// TIA Portal project "练习一视觉分拣" (V16)

(* hardware
DEVICE "S7-1200 station_1"  S7-1200 Station
   slot 0: "Rack_0"  S7-1200 Rack  Rack  V1.0
   slot 1: "PLC_1"  CPU 1214C DC/DC/Rly  6ES7 214-1HG40-0XB0  V4.4
DEVICE "HMI_1"  KTP700 Basic PN
   slot 0: "HMI_1"  KTP700 Basic PN  6AV2 123-2GB03-0AX0  16.0.0.0
   slot 1: "HMI_RT_1"  KTP700 Basic PN  6AV2 123-2GB03-0AX0  16.0.0.0
   slot 5: "HMI_1.IE_CP_1"  PROFINET Interface  16.0.0.0
      slot 1: "PROFINET Interface_1"  PROFINET Interface
         slot 1: "Port_1"  Port
*)

// ===== PLC "PLC_1"  CPU 1214C DC/DC/Rly =====

VAR_GLOBAL   // PLC tag table "默认变量表"
   "System_Byte" AT %MB1 : Byte;
   "FirstScan" AT %M1.0 : Bool;
   "DiagStatusUpdate" AT %M1.1 : Bool;
   "AlwaysTRUE" AT %M1.2 : Bool;
   "AlwaysFALSE" AT %M1.3 : Bool;
   "Clock_Byte" AT %MB0 : Byte;
   "Clock_10Hz" AT %M0.0 : Bool;
   "Clock_5Hz" AT %M0.1 : Bool;
   "Clock_2.5Hz" AT %M0.2 : Bool;
   "Clock_2Hz" AT %M0.3 : Bool;
   "Clock_1.25Hz" AT %M0.4 : Bool;
   "Clock_1Hz" AT %M0.5 : Bool;
   "Clock_0.625Hz" AT %M0.6 : Bool;
   "Clock_0.5Hz" AT %M0.7 : Bool;
END_VAR

VAR_GLOBAL   // PLC tag table "io"
   "启动信号" AT %I0.0 : Bool;
   "停止信号" AT %I0.1 : Bool;
   "复位信号" AT %I0.2 : Bool;
   "急停信号" AT %I0.3 : Bool;
   "左转到位i传感器" AT %I0.5 : Bool;
   "右转到位传感器" AT %I0.6 : Bool;
   "直行到位传感器" AT %I0.7 : Bool;
   "手动开关" AT %I1.0 : Bool;
   "自动开关" AT %I1.1 : Bool;
   "运行指示灯" AT %Q0.0 : Bool;
   "停止指示灯" AT %Q0.1 : Bool;
   "复位指示灯" AT %Q0.2 : Bool;
   "供料输送机" AT %Q0.3 : Bool;
   "直行电机" AT %Q0.4 : Bool;
   "左转电机" AT %Q0.5 : Bool;
   "右转电机" AT %Q0.6 : Bool;
   "产品原料分拣机" AT %Q0.7 : Bool;
   "产品基座分拣机" AT %Q1.0 : Bool;
   "产品盖分拣机" AT %Q1.1 : Bool;
   "物料生成器" AT %Q1.2 : Bool;
   "阻挡器" AT %Q1.3 : Bool;
   "视觉相机" AT %ID30 : DInt;
END_VAR

DATA_BLOCK "核心功能区"   // DB1
{ S7_Optimized_Access := 'TRUE' }
VERSION : 0.1
   VAR
      核心程序步 : Int;
      中间变量1 : Bool;
      中间变量2 : Bool;
      中间变量3 : Bool;
   END_VAR
BEGIN
END_DATA_BLOCK

DATA_BLOCK "FC程序视觉核心分拣区DB"   // DB2
{ S7_Optimized_Access := 'TRUE' }
VERSION : 0.1
   VAR
      FC核心程序编写 : Int;
      FC中间变量1 : Bool;
      FC中间变量2 : Bool;
      FC中间变量3 : Bool;
   END_VAR
BEGIN
END_DATA_BLOCK

DATA_BLOCK "主程序"   // DB3
{ S7_Optimized_Access := 'TRUE' }
VERSION : 0.1
   VAR
      核心程序步 : Int;
      复位标志位 : Bool;
      启动信号 : Bool;
      停止信号 : Bool;
      复位信号 : Bool;
      "手/自动切换" : Bool;
      急停信号 : Bool := true;
      中间变量1 : Bool;
      中间变量2 : Bool;
      中间变量3 : Bool;
      中间变量4 : Bool;
      运行模式 : Int;
   END_VAR
BEGIN
END_DATA_BLOCK

// folder: 01_核心分拣区

DATA_BLOCK "FB视觉分拣核心区_DB"   // DB4
{ S7_Optimized_Access := 'TRUE' }
VERSION : 0.1
// stored: InstanceOfName FB视觉分拣核心区
"FB视觉分拣核心区"
BEGIN
END_DATA_BLOCK

// folder: 02_自动运行模式

DATA_BLOCK "自动运行模式_DB"   // DB5
{ S7_Optimized_Access := 'TRUE' }
VERSION : 0.1
// stored: InstanceOfName 自动运行模式
"自动运行模式"
BEGIN
END_DATA_BLOCK

// folder: 03_手动运行模式

DATA_BLOCK "手动运行模式_DB"   // DB6
{ S7_Optimized_Access := 'TRUE' }
VERSION : 0.1
// stored: InstanceOfName 手动运行模式
"手动运行模式"
BEGIN
END_DATA_BLOCK

DATA_BLOCK "FB视觉分拣核心区_DB_1"   // DB7
{ S7_Optimized_Access := 'TRUE' }
VERSION : 0.1
// stored: InstanceOfName FB视觉分拣核心区
"FB视觉分拣核心区"
BEGIN
END_DATA_BLOCK

// folder: 04_系统急停

DATA_BLOCK "系统急停_DB"   // DB8
{ S7_Optimized_Access := 'TRUE' }
VERSION : 0.1
// stored: InstanceOfName 系统急停
"系统急停"
BEGIN
END_DATA_BLOCK

// folder: 05_系统复位

DATA_BLOCK "系统复位_DB"   // DB9
{ S7_Optimized_Access := 'TRUE' }
VERSION : 0.1
// stored: InstanceOfName 系统复位
"系统复位"
BEGIN
END_DATA_BLOCK

DATA_BLOCK "FB视觉分拣核心区_DB_2"   // DB10
{ S7_Optimized_Access := 'TRUE' }
VERSION : 0.1
// stored: InstanceOfName FB视觉分拣核心区
"FB视觉分拣核心区"
BEGIN
END_DATA_BLOCK

// folder: (top level)

FUNCTION "视觉分拣核心区" : Void   // FC1, LAD
{ S7_Optimized_Access := 'TRUE' }
VERSION : 0.1
   VAR_INPUT
      视觉相机传感器 : DWord;
      直行到传感器 : Bool;
      左转到位传感器 : Bool;
      右转到位传感器 : Bool;
   END_VAR
   VAR_OUTPUT
      直行电机 : Bool;
      左转电机 : Bool;
      右转电机 : Bool;
   END_VAR
   VAR_IN_OUT
      核心分拣区程序步 : Int;
   END_VAR
   VAR_TEMP   // added for the SCL form of the ladder/FBD networks
      _w1 : Bool;
   END_VAR
BEGIN

REGION Network 1: 物料分辨
   // 将输入数据给调为形参，将检查到的数据，给传递给，核心功能区
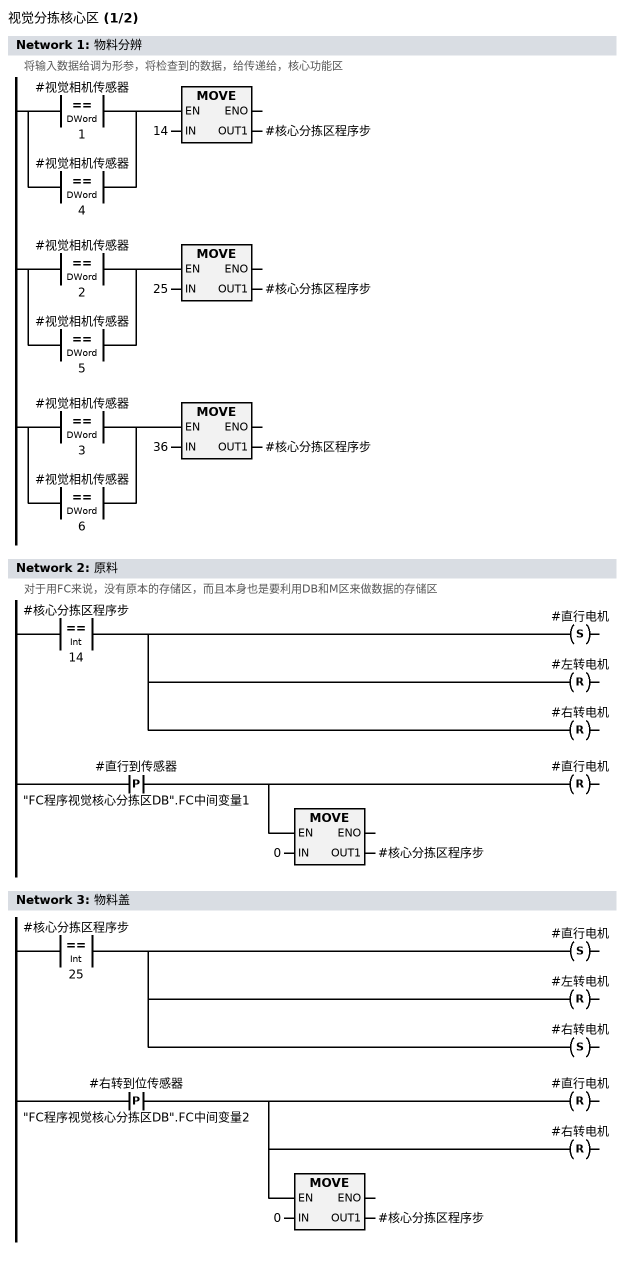
   RUNG wire#powerrail
      { S7_Templates := "SrcType := DWord" } EQ_Contact(in1 := #视觉相机传感器, in2 := 1)
      wire#w1
      Move(in := 14, out1 => #核心分拣区程序步)
   END_RUNG
   RUNG wire#powerrail
      { S7_Templates := "SrcType := DWord" } EQ_Contact(in1 := #视觉相机传感器, in2 := 4)
   END_RUNG wire#w1
   RUNG wire#powerrail
      { S7_Templates := "SrcType := DWord" } EQ_Contact(in1 := #视觉相机传感器, in2 := 2)
      wire#w2
      Move(in := 25, out1 => #核心分拣区程序步)
   END_RUNG
   RUNG wire#powerrail
      { S7_Templates := "SrcType := DWord" } EQ_Contact(in1 := #视觉相机传感器, in2 := 5)
   END_RUNG wire#w2
   RUNG wire#powerrail
      { S7_Templates := "SrcType := DWord" } EQ_Contact(in1 := #视觉相机传感器, in2 := 3)
      wire#w3
      Move(in := 36, out1 => #核心分拣区程序步)
   END_RUNG
   RUNG wire#powerrail
      { S7_Templates := "SrcType := DWord" } EQ_Contact(in1 := #视觉相机传感器, in2 := 6)
   END_RUNG wire#w3
   // the same network as SCL:
   IF (#视觉相机传感器 = 1) OR (#视觉相机传感器 = 4) THEN #核心分拣区程序步 := 14; END_IF;
   IF (#视觉相机传感器 = 2) OR (#视觉相机传感器 = 5) THEN #核心分拣区程序步 := 25; END_IF;
   IF (#视觉相机传感器 = 3) OR (#视觉相机传感器 = 6) THEN #核心分拣区程序步 := 36; END_IF;
END_REGION

REGION Network 2: 原料
   // 对于用FC来说，没有原本的存储区，而且本身也是要利用DB和M区来做数据的存储区
   RUNG wire#powerrail
      { S7_Templates := "SrcType := Int" } EQ_Contact(in1 := #核心分拣区程序步, in2 := 14)
      wire#w1
      S_Coil( #直行电机 )
   END_RUNG
   RUNG wire#w1
      R_Coil( #左转电机 )
   END_RUNG
   RUNG wire#w1
      R_Coil( #右转电机 )
   END_RUNG
   RUNG wire#powerrail
      P_Contact(operand := #直行到传感器, bit := "FC程序视觉核心分拣区DB".FC中间变量1)
      wire#w2
      R_Coil( #直行电机 )
   END_RUNG
   RUNG wire#w2
      Move(in := 0, out1 => #核心分拣区程序步)
   END_RUNG
   // the same network as SCL:
   IF #核心分拣区程序步 = 14 THEN
       #直行电机 := TRUE;
       #左转电机 := FALSE;
       #右转电机 := FALSE;
   END_IF;
   #_w1 := #直行到传感器 AND NOT "FC程序视觉核心分拣区DB".FC中间变量1;   // rising edge of #直行到传感器
   "FC程序视觉核心分拣区DB".FC中间变量1 := #直行到传感器;
   IF #_w1 THEN
       #直行电机 := FALSE;
       #核心分拣区程序步 := 0;
   END_IF;
END_REGION

REGION Network 3: 物料盖
   RUNG wire#powerrail
      { S7_Templates := "SrcType := Int" } EQ_Contact(in1 := #核心分拣区程序步, in2 := 25)
      wire#w1
      S_Coil( #直行电机 )
   END_RUNG
   RUNG wire#w1
      R_Coil( #左转电机 )
   END_RUNG
   RUNG wire#w1
      S_Coil( #右转电机 )
   END_RUNG
   RUNG wire#powerrail
      P_Contact(operand := #右转到位传感器, bit := "FC程序视觉核心分拣区DB".FC中间变量2)
      wire#w2
      R_Coil( #直行电机 )
   END_RUNG
   RUNG wire#w2
      R_Coil( #右转电机 )
   END_RUNG
   RUNG wire#w2
      Move(in := 0, out1 => #核心分拣区程序步)
   END_RUNG
   // the same network as SCL:
   IF #核心分拣区程序步 = 25 THEN
       #直行电机 := TRUE;
       #左转电机 := FALSE;
       #右转电机 := TRUE;
   END_IF;
   #_w1 := #右转到位传感器 AND NOT "FC程序视觉核心分拣区DB".FC中间变量2;   // rising edge of #右转到位传感器
   "FC程序视觉核心分拣区DB".FC中间变量2 := #右转到位传感器;
   IF #_w1 THEN
       #直行电机 := FALSE;
       #右转电机 := FALSE;
       #核心分拣区程序步 := 0;
   END_IF;
END_REGION

REGION Network 4: 物料基座
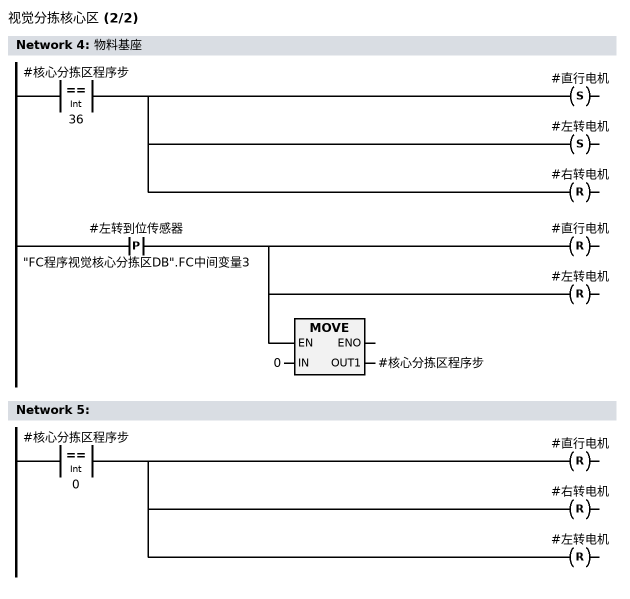
   RUNG wire#powerrail
      { S7_Templates := "SrcType := Int" } EQ_Contact(in1 := #核心分拣区程序步, in2 := 36)
      wire#w1
      S_Coil( #直行电机 )
   END_RUNG
   RUNG wire#w1
      S_Coil( #左转电机 )
   END_RUNG
   RUNG wire#w1
      R_Coil( #右转电机 )
   END_RUNG
   RUNG wire#powerrail
      P_Contact(operand := #左转到位传感器, bit := "FC程序视觉核心分拣区DB".FC中间变量3)
      wire#w2
      R_Coil( #直行电机 )
   END_RUNG
   RUNG wire#w2
      R_Coil( #左转电机 )
   END_RUNG
   RUNG wire#w2
      Move(in := 0, out1 => #核心分拣区程序步)
   END_RUNG
   // the same network as SCL:
   IF #核心分拣区程序步 = 36 THEN
       #直行电机 := TRUE;
       #左转电机 := TRUE;
       #右转电机 := FALSE;
   END_IF;
   #_w1 := #左转到位传感器 AND NOT "FC程序视觉核心分拣区DB".FC中间变量3;   // rising edge of #左转到位传感器
   "FC程序视觉核心分拣区DB".FC中间变量3 := #左转到位传感器;
   IF #_w1 THEN
       #直行电机 := FALSE;
       #左转电机 := FALSE;
       #核心分拣区程序步 := 0;
   END_IF;
END_REGION

REGION Network 5
   RUNG wire#powerrail
      { S7_Templates := "SrcType := Int" } EQ_Contact(in1 := #核心分拣区程序步, in2 := 0)
      wire#w1
      R_Coil( #直行电机 )
   END_RUNG
   RUNG wire#w1
      R_Coil( #右转电机 )
   END_RUNG
   RUNG wire#w1
      R_Coil( #左转电机 )
   END_RUNG
   // the same network as SCL:
   IF #核心分拣区程序步 = 0 THEN
       #直行电机 := FALSE;
       #右转电机 := FALSE;
       #左转电机 := FALSE;
   END_IF;
END_REGION
END_FUNCTION

FUNCTION "MHJ-PLC-Lab-Function-S71200" : Void   // FC9000, SCL
{ S7_Optimized_Access := 'TRUE' }
VERSION : 0.1
   VAR_TEMP
      rdTimeReturn : Int;
      outputTime : DTL;
      SyncVal : Byte;
      forVal : Int;
      forVal_2 : Int;
      Value : Byte;
   END_VAR
   VAR CONSTANT
      CompVal : Byte := 16#34;
      Value_01 : Byte := 16#11;
      Value_01_DW : DWord := 16#A165_D992;
      Value_02_DW : DWord := 16#58BE_4401;
   END_VAR
BEGIN

   #Value:=PEEK(area := 16#82,
        dbNumber := 0,
        byteOffset := 511);
   #Value := #Value + 1;

   POKE(area := 16#82,
        dbNumber := 0,
        byteOffset := 511,
        value := #Value);

   POKE(area:=16#81,
        dbNumber:=0,
        byteOffset:=1016,
        value:=#Value_01_DW);
   POKE(area := 16#81,
        dbNumber := 0,
        byteOffset := 1020,
        value := #Value_02_DW);

   POKE(area := 16#81,
        dbNumber := 0,
        byteOffset := 511,
        value := B#16#00);

   FOR #forVal := 0 TO 120 DO
       FOR #forVal_2:=0 TO 10 DO
           #rdTimeReturn:=RD_SYS_T(#outputTime);
           #rdTimeReturn := WR_SYS_T(#outputTime);
           #rdTimeReturn := RD_SYS_T(#outputTime);
           #rdTimeReturn := WR_SYS_T(#outputTime);
       END_FOR;
       #SyncVal:= PEEK(area := 16#81,
                      dbNumber := 0,
                      byteOffset := 511);
       IF #SyncVal = #CompVal THEN
          GOTO M_1;
       END_IF;
   END_FOR;
   RETURN;

   M_1:
   POKE(area := 16#81,
        dbNumber := 0,
        byteOffset := 511,
        value := B#16#0);
END_FUNCTION

ORGANIZATION_BLOCK "Main"   // OB1, LAD, ProgramCycle
TITLE = "Main Program Sweep (Cycle)"
{ S7_Optimized_Access := 'TRUE' }
VERSION : 0.1
   VAR_INPUT
      Initial_Call : Bool;   // Initial call of this OB
      Remanence : Bool;   // =True, if remanent data are available
   END_VAR
   VAR_TEMP   // added for the SCL form of the ladder/FBD networks
      _w1 : Bool;
      _w2 : Bool;
      _w3 : Bool;
      _w4 : Bool;
   END_VAR
BEGIN

REGION Network 1
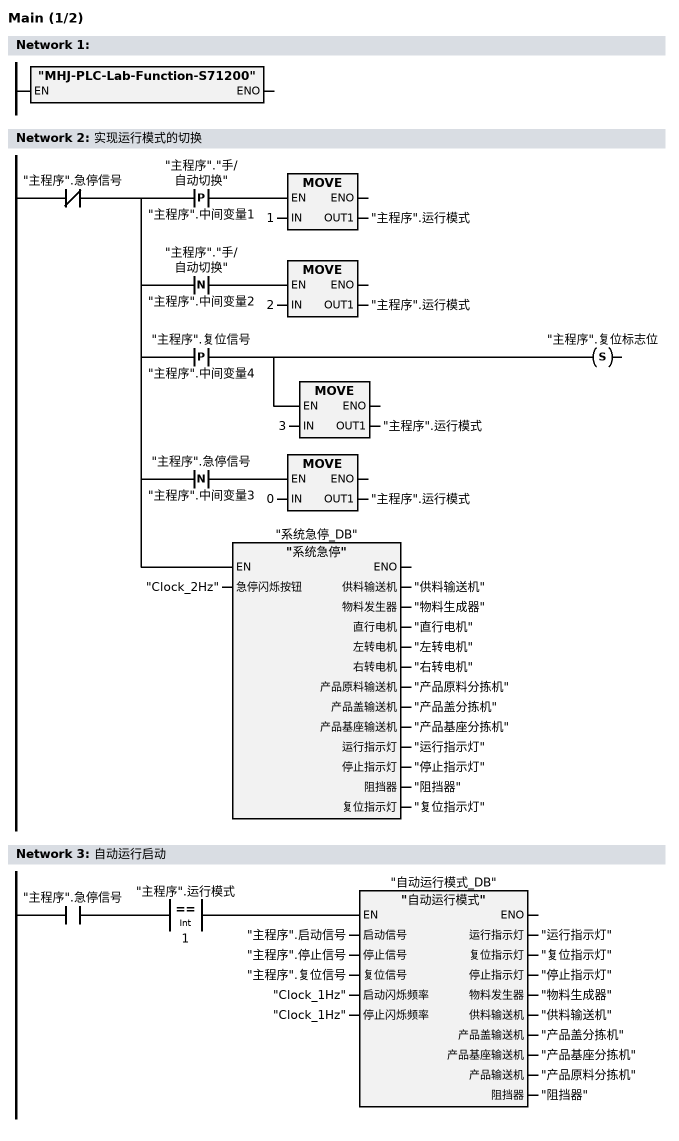
   RUNG wire#powerrail
      "MHJ-PLC-Lab-Function-S71200"()
   END_RUNG
   // the same network as SCL:
   "MHJ-PLC-Lab-Function-S71200"();
END_REGION

REGION Network 2: 实现运行模式的切换
   RUNG wire#powerrail
      I_Contact( "主程序".急停信号 )
      wire#w1
      P_Contact(operand := "主程序"."手/自动切换", bit := "主程序".中间变量1)
      Move(in := 1, out1 => "主程序".运行模式)
   END_RUNG
   RUNG wire#w1
      N_Contact(operand := "主程序"."手/自动切换", bit := "主程序".中间变量2)
      Move(in := 2, out1 => "主程序".运行模式)
   END_RUNG
   RUNG wire#w1
      P_Contact(operand := "主程序".复位信号, bit := "主程序".中间变量4)
      wire#w2
      S_Coil( "主程序".复位标志位 )
   END_RUNG
   RUNG wire#w2
      Move(in := 3, out1 => "主程序".运行模式)
   END_RUNG
   RUNG wire#w1
      N_Contact(operand := "主程序".急停信号, bit := "主程序".中间变量3)
      Move(in := 0, out1 => "主程序".运行模式)
   END_RUNG
   RUNG wire#w1
      "系统急停_DB"(急停闪烁按钮 := "Clock_2Hz", 供料输送机 => "供料输送机", 物料发生器 => "物料生成器", 直行电机 => "直行电机", 左转电机 => "左转电机", 右转电机 => "右转电机", 产品原料输送机 => "产品原料分拣机", 产品盖输送机 => "产品盖分拣机", 产品基座输送机 => "产品基座分拣机", 运行指示灯 => "运行指示灯", 停止指示灯 => "停止指示灯", 阻挡器 => "阻挡器", 复位指示灯 => "复位指示灯")
   END_RUNG
   // the same network as SCL:
   #_w1 := NOT "主程序".急停信号 AND "主程序"."手/自动切换" AND NOT "主程序".中间变量1;   // rising edge of "主程序"."手/自动切换"
   "主程序".中间变量1 := "主程序"."手/自动切换";
   IF #_w1 THEN "主程序".运行模式 := 1; END_IF;
   #_w2 := NOT "主程序".急停信号 AND NOT "主程序"."手/自动切换" AND "主程序".中间变量2;   // falling edge of "主程序"."手/自动切换"
   "主程序".中间变量2 := "主程序"."手/自动切换";
   IF #_w2 THEN "主程序".运行模式 := 2; END_IF;
   #_w3 := NOT "主程序".急停信号 AND "主程序".复位信号 AND NOT "主程序".中间变量4;   // rising edge of "主程序".复位信号
   "主程序".中间变量4 := "主程序".复位信号;
   IF #_w3 THEN
       "主程序".复位标志位 := TRUE;
       "主程序".运行模式 := 3;
   END_IF;
   #_w4 := NOT "主程序".急停信号 AND NOT "主程序".急停信号 AND "主程序".中间变量3;   // falling edge of "主程序".急停信号
   "主程序".中间变量3 := "主程序".急停信号;
   IF #_w4 THEN "主程序".运行模式 := 0; END_IF;
   IF NOT "主程序".急停信号 THEN
       "系统急停_DB"(急停闪烁按钮 := "Clock_2Hz",   // "系统急停"
                 供料输送机 => "供料输送机",
                 物料发生器 => "物料生成器",
                 直行电机 => "直行电机",
                 左转电机 => "左转电机",
                 右转电机 => "右转电机",
                 产品原料输送机 => "产品原料分拣机",
                 产品盖输送机 => "产品盖分拣机",
                 产品基座输送机 => "产品基座分拣机",
                 运行指示灯 => "运行指示灯",
                 停止指示灯 => "停止指示灯",
                 阻挡器 => "阻挡器",
                 复位指示灯 => "复位指示灯");
   END_IF;
END_REGION

REGION Network 3: 自动运行启动
   RUNG wire#powerrail
      Contact( "主程序".急停信号 )
      { S7_Templates := "SrcType := Int" } EQ_Contact(in1 := "主程序".运行模式, in2 := 1)
      "自动运行模式_DB"(启动信号 := "主程序".启动信号, 停止信号 := "主程序".停止信号, 复位信号 := "主程序".复位信号, 启动闪烁频率 := "Clock_1Hz", 停止闪烁频率 := "Clock_1Hz", 运行指示灯 => "运行指示灯", 复位指示灯 => "复位指示灯", 停止指示灯 => "停止指示灯", 物料发生器 => "物料生成器", 供料输送机 => "供料输送机", 产品盖输送机 => "产品盖分拣机", 产品基座输送机 => "产品基座分拣机", 产品输送机 => "产品原料分拣机", 阻挡器 => "阻挡器")
   END_RUNG
   // the same network as SCL:
   IF "主程序".急停信号 AND ("主程序".运行模式 = 1) THEN
       "自动运行模式_DB"(启动信号 := "主程序".启动信号,   // "自动运行模式"
                   停止信号 := "主程序".停止信号,
                   复位信号 := "主程序".复位信号,
                   启动闪烁频率 := "Clock_1Hz",
                   停止闪烁频率 := "Clock_1Hz",
                   运行指示灯 => "运行指示灯",
                   复位指示灯 => "复位指示灯",
                   停止指示灯 => "停止指示灯",
                   物料发生器 => "物料生成器",
                   供料输送机 => "供料输送机",
                   产品盖输送机 => "产品盖分拣机",
                   产品基座输送机 => "产品基座分拣机",
                   产品输送机 => "产品原料分拣机",
                   阻挡器 => "阻挡器");
   END_IF;
END_REGION

REGION Network 4: 手动运行启动
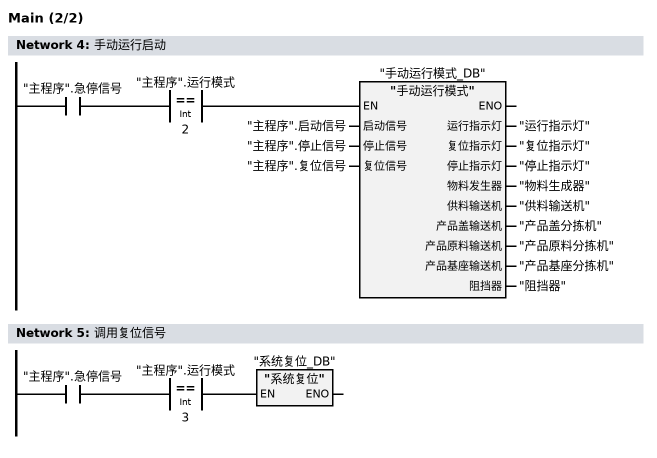
   RUNG wire#powerrail
      Contact( "主程序".急停信号 )
      { S7_Templates := "SrcType := Int" } EQ_Contact(in1 := "主程序".运行模式, in2 := 2)
      "手动运行模式_DB"(启动信号 := "主程序".启动信号, 停止信号 := "主程序".停止信号, 复位信号 := "主程序".复位信号, 运行指示灯 => "运行指示灯", 复位指示灯 => "复位指示灯", 停止指示灯 => "停止指示灯", 物料发生器 => "物料生成器", 供料输送机 => "供料输送机", 产品盖输送机 => "产品盖分拣机", 产品原料输送机 => "产品原料分拣机", 产品基座输送机 => "产品基座分拣机", 阻挡器 => "阻挡器")
   END_RUNG
   // the same network as SCL:
   IF "主程序".急停信号 AND ("主程序".运行模式 = 2) THEN
       "手动运行模式_DB"(启动信号 := "主程序".启动信号,   // "手动运行模式"
                   停止信号 := "主程序".停止信号,
                   复位信号 := "主程序".复位信号,
                   运行指示灯 => "运行指示灯",
                   复位指示灯 => "复位指示灯",
                   停止指示灯 => "停止指示灯",
                   物料发生器 => "物料生成器",
                   供料输送机 => "供料输送机",
                   产品盖输送机 => "产品盖分拣机",
                   产品原料输送机 => "产品原料分拣机",
                   产品基座输送机 => "产品基座分拣机",
                   阻挡器 => "阻挡器");
   END_IF;
END_REGION

REGION Network 5: 调用复位信号
   RUNG wire#powerrail
      Contact( "主程序".急停信号 )
      { S7_Templates := "SrcType := Int" } EQ_Contact(in1 := "主程序".运行模式, in2 := 3)
      "系统复位_DB"()
   END_RUNG
   // the same network as SCL:
   IF "主程序".急停信号 AND ("主程序".运行模式 = 3) THEN
       "系统复位_DB"();   // "系统复位"
   END_IF;
END_REGION
END_ORGANIZATION_BLOCK

// folder: 01_核心分拣区

FUNCTION_BLOCK "FB视觉分拣核心区"   // FB1, LAD
{ S7_Optimized_Access := 'TRUE' }
VERSION : 0.1
   VAR_INPUT
      视觉相机 : DWord;
      直行到位传感器 : Bool;
      左转到位传感器 : Bool;
      右转到位传感器 : Bool;
   END_VAR
   VAR_OUTPUT
      直行电机 : Bool;
      左转电机 : Bool;
      右转电机 : Bool;
   END_VAR
   VAR_IN_OUT
      FB程序步 : Int;
   END_VAR
   VAR
      中间变量1 : Bool;
      中间变量2 : Bool;
      中间变量3 : Bool;
   END_VAR
   VAR_TEMP   // added for the SCL form of the ladder/FBD networks
      _w1 : Bool;
   END_VAR
BEGIN

REGION Network 1: 物料分辨
   // 将输入数据给调为形参，将检查到的数据，给传递给，核心功能区
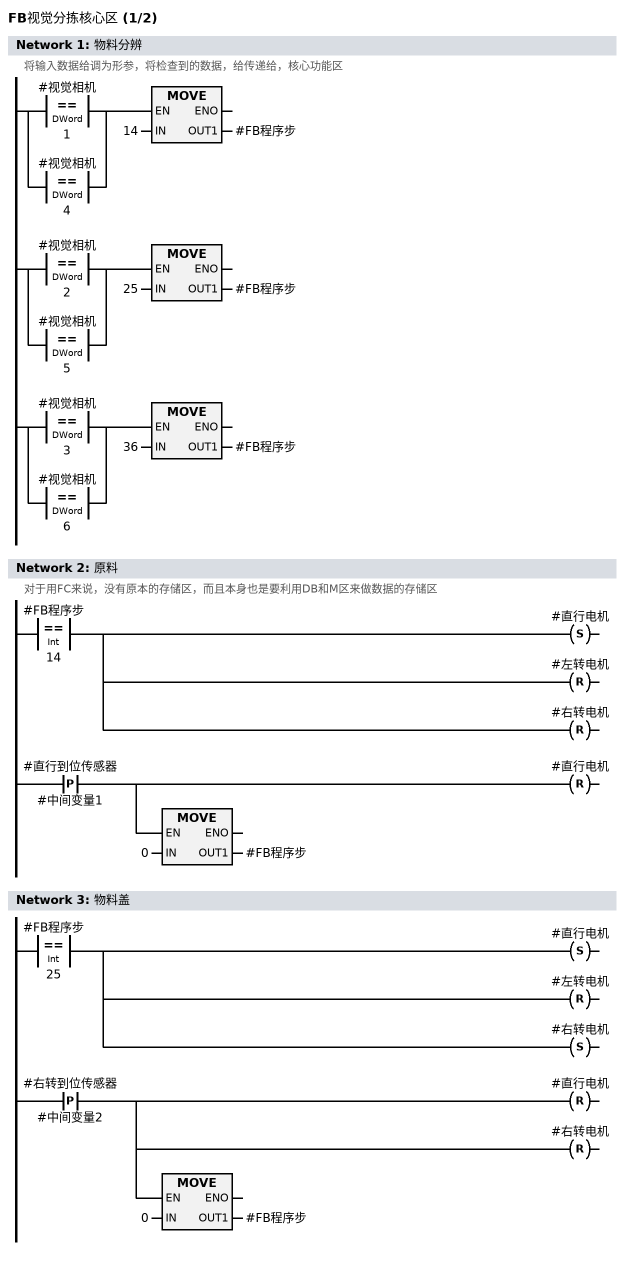
   RUNG wire#powerrail
      { S7_Templates := "SrcType := DWord" } EQ_Contact(in1 := #视觉相机, in2 := 1)
      wire#w1
      Move(in := 14, out1 => #FB程序步)
   END_RUNG
   RUNG wire#powerrail
      { S7_Templates := "SrcType := DWord" } EQ_Contact(in1 := #视觉相机, in2 := 4)
   END_RUNG wire#w1
   RUNG wire#powerrail
      { S7_Templates := "SrcType := DWord" } EQ_Contact(in1 := #视觉相机, in2 := 2)
      wire#w2
      Move(in := 25, out1 => #FB程序步)
   END_RUNG
   RUNG wire#powerrail
      { S7_Templates := "SrcType := DWord" } EQ_Contact(in1 := #视觉相机, in2 := 5)
   END_RUNG wire#w2
   RUNG wire#powerrail
      { S7_Templates := "SrcType := DWord" } EQ_Contact(in1 := #视觉相机, in2 := 3)
      wire#w3
      Move(in := 36, out1 => #FB程序步)
   END_RUNG
   RUNG wire#powerrail
      { S7_Templates := "SrcType := DWord" } EQ_Contact(in1 := #视觉相机, in2 := 6)
   END_RUNG wire#w3
   // the same network as SCL:
   IF (#视觉相机 = 1) OR (#视觉相机 = 4) THEN #FB程序步 := 14; END_IF;
   IF (#视觉相机 = 2) OR (#视觉相机 = 5) THEN #FB程序步 := 25; END_IF;
   IF (#视觉相机 = 3) OR (#视觉相机 = 6) THEN #FB程序步 := 36; END_IF;
END_REGION

REGION Network 2: 原料
   // 对于用FC来说，没有原本的存储区，而且本身也是要利用DB和M区来做数据的存储区
   RUNG wire#powerrail
      { S7_Templates := "SrcType := Int" } EQ_Contact(in1 := #FB程序步, in2 := 14)
      wire#w1
      S_Coil( #直行电机 )
   END_RUNG
   RUNG wire#w1
      R_Coil( #左转电机 )
   END_RUNG
   RUNG wire#w1
      R_Coil( #右转电机 )
   END_RUNG
   RUNG wire#powerrail
      P_Contact(operand := #直行到位传感器, bit := #中间变量1)
      wire#w2
      R_Coil( #直行电机 )
   END_RUNG
   RUNG wire#w2
      Move(in := 0, out1 => #FB程序步)
   END_RUNG
   // the same network as SCL:
   IF #FB程序步 = 14 THEN
       #直行电机 := TRUE;
       #左转电机 := FALSE;
       #右转电机 := FALSE;
   END_IF;
   #_w1 := #直行到位传感器 AND NOT #中间变量1;   // rising edge of #直行到位传感器
   #中间变量1 := #直行到位传感器;
   IF #_w1 THEN
       #直行电机 := FALSE;
       #FB程序步 := 0;
   END_IF;
END_REGION

REGION Network 3: 物料盖
   RUNG wire#powerrail
      { S7_Templates := "SrcType := Int" } EQ_Contact(in1 := #FB程序步, in2 := 25)
      wire#w1
      S_Coil( #直行电机 )
   END_RUNG
   RUNG wire#w1
      R_Coil( #左转电机 )
   END_RUNG
   RUNG wire#w1
      S_Coil( #右转电机 )
   END_RUNG
   RUNG wire#powerrail
      P_Contact(operand := #右转到位传感器, bit := #中间变量2)
      wire#w2
      R_Coil( #直行电机 )
   END_RUNG
   RUNG wire#w2
      R_Coil( #右转电机 )
   END_RUNG
   RUNG wire#w2
      Move(in := 0, out1 => #FB程序步)
   END_RUNG
   // the same network as SCL:
   IF #FB程序步 = 25 THEN
       #直行电机 := TRUE;
       #左转电机 := FALSE;
       #右转电机 := TRUE;
   END_IF;
   #_w1 := #右转到位传感器 AND NOT #中间变量2;   // rising edge of #右转到位传感器
   #中间变量2 := #右转到位传感器;
   IF #_w1 THEN
       #直行电机 := FALSE;
       #右转电机 := FALSE;
       #FB程序步 := 0;
   END_IF;
END_REGION

REGION Network 4: 物料基座
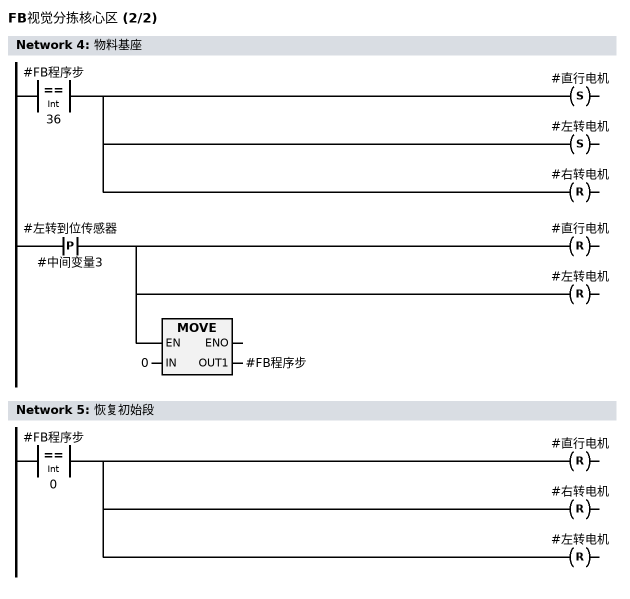
   RUNG wire#powerrail
      { S7_Templates := "SrcType := Int" } EQ_Contact(in1 := #FB程序步, in2 := 36)
      wire#w1
      S_Coil( #直行电机 )
   END_RUNG
   RUNG wire#w1
      S_Coil( #左转电机 )
   END_RUNG
   RUNG wire#w1
      R_Coil( #右转电机 )
   END_RUNG
   RUNG wire#powerrail
      P_Contact(operand := #左转到位传感器, bit := #中间变量3)
      wire#w2
      R_Coil( #直行电机 )
   END_RUNG
   RUNG wire#w2
      R_Coil( #左转电机 )
   END_RUNG
   RUNG wire#w2
      Move(in := 0, out1 => #FB程序步)
   END_RUNG
   // the same network as SCL:
   IF #FB程序步 = 36 THEN
       #直行电机 := TRUE;
       #左转电机 := TRUE;
       #右转电机 := FALSE;
   END_IF;
   #_w1 := #左转到位传感器 AND NOT #中间变量3;   // rising edge of #左转到位传感器
   #中间变量3 := #左转到位传感器;
   IF #_w1 THEN
       #直行电机 := FALSE;
       #左转电机 := FALSE;
       #FB程序步 := 0;
   END_IF;
END_REGION

REGION Network 5: 恢复初始段
   RUNG wire#powerrail
      { S7_Templates := "SrcType := Int" } EQ_Contact(in1 := #FB程序步, in2 := 0)
      wire#w1
      R_Coil( #直行电机 )
   END_RUNG
   RUNG wire#w1
      R_Coil( #右转电机 )
   END_RUNG
   RUNG wire#w1
      R_Coil( #左转电机 )
   END_RUNG
   // the same network as SCL:
   IF #FB程序步 = 0 THEN
       #直行电机 := FALSE;
       #右转电机 := FALSE;
       #左转电机 := FALSE;
   END_IF;
END_REGION
END_FUNCTION_BLOCK

// folder: 02_自动运行模式

FUNCTION_BLOCK "自动运行模式"   // FB2, LAD
{ S7_Optimized_Access := 'TRUE' }
VERSION : 0.1
   VAR_INPUT
      启动信号 : Bool;
      停止信号 : Bool;
      复位信号 : Bool;
      启动闪烁频率 : Bool;
      停止闪烁频率 : Bool;
   END_VAR
   VAR_OUTPUT
      运行指示灯 : Bool;
      复位指示灯 : Bool;
      停止指示灯 : Bool;
      物料发生器 : Bool;
      供料输送机 : Bool;
      产品盖输送机 : Bool;
      产品基座输送机 : Bool;
      产品输送机 : Bool;
      阻挡器 : Bool;
   END_VAR
   VAR
      自动启动运行中 : Bool;
      自动启动运行完成 : Bool;
      自动关闭运行中 : Bool;
      自动关闭完成 : Bool;
      中间变量1 : Bool;
      中间变量2 : Bool;
      中间变量3 : Bool;
      中间变量4 : Bool;
      中间变量5 : Bool;
      IEC_Timer_0_Instance_01 : TON_TIME;
      IEC_Timer_0_Instance_02 : TON_TIME;
   END_VAR
   VAR_TEMP   // added for the SCL form of the ladder/FBD networks
      _w1 : Bool;
      _w2 : Bool;
   END_VAR
BEGIN

REGION Network 1: 启动分拣输送机
   // 开始启动完成之前，需要将三个运输机发动起来，而且在开始启动的时候要保持绿灯闪烁5是，之后开始产生物料和运输物料。因为在我们在子程序中编写，不太好应用编程闪烁，
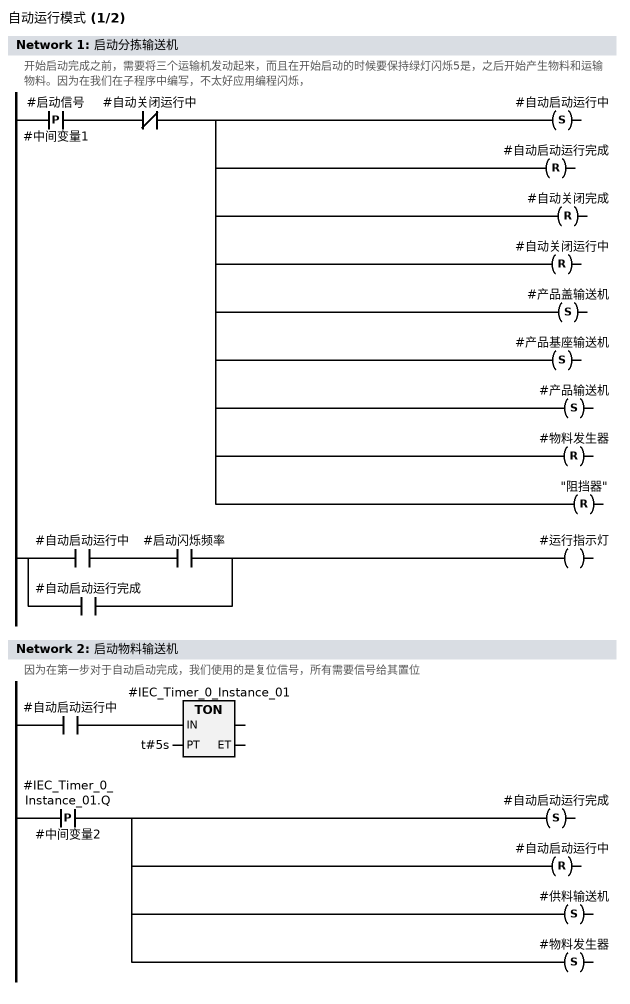
   RUNG wire#powerrail
      P_Contact(operand := #启动信号, bit := #中间变量1)
      I_Contact( #自动关闭运行中 )
      wire#w1
      S_Coil( #自动启动运行中 )
   END_RUNG
   RUNG wire#w1
      R_Coil( #自动启动运行完成 )
   END_RUNG
   RUNG wire#w1
      R_Coil( #自动关闭完成 )
   END_RUNG
   RUNG wire#w1
      R_Coil( #自动关闭运行中 )
   END_RUNG
   RUNG wire#w1
      S_Coil( #产品盖输送机 )
   END_RUNG
   RUNG wire#w1
      S_Coil( #产品基座输送机 )
   END_RUNG
   RUNG wire#w1
      S_Coil( #产品输送机 )
   END_RUNG
   RUNG wire#w1
      R_Coil( #物料发生器 )
   END_RUNG
   RUNG wire#w1
      R_Coil( "阻挡器" )
   END_RUNG
   RUNG wire#powerrail
      Contact( #自动启动运行中 )
      Contact( #启动闪烁频率 )
      wire#w2
      Coil( #运行指示灯 )
   END_RUNG
   RUNG wire#powerrail
      Contact( #自动启动运行完成 )
   END_RUNG wire#w2
   // the same network as SCL:
   #_w1 := #启动信号 AND NOT #中间变量1;   // rising edge of #启动信号
   #中间变量1 := #启动信号;
   IF #_w1 AND NOT #自动关闭运行中 THEN
       #自动启动运行中 := TRUE;
       #自动启动运行完成 := FALSE;
       #自动关闭完成 := FALSE;
   END_IF;
   #_w2 := #_w1 AND NOT #自动关闭运行中;
   IF #_w2 THEN
       #自动关闭运行中 := FALSE;
       #产品盖输送机 := TRUE;
       #产品基座输送机 := TRUE;
       #产品输送机 := TRUE;
       #物料发生器 := FALSE;
       "阻挡器" := FALSE;
   END_IF;
   #运行指示灯 := (#自动启动运行中 AND #启动闪烁频率) OR #自动启动运行完成;
END_REGION

REGION Network 2: 启动物料输送机
   // 因为在第一步对于自动启动完成，我们使用的是复位信号，所有需要信号给其置位
   #IEC_Timer_0_Instance_01(IN := #自动启动运行中, PT := t#5s);   // TON
   #_w1 := #IEC_Timer_0_Instance_01.Q AND NOT #中间变量2;   // rising edge of #IEC_Timer_0_Instance_01.Q
   #中间变量2 := #IEC_Timer_0_Instance_01.Q;
   IF #_w1 THEN
       #自动启动运行完成 := TRUE;
       #自动启动运行中 := FALSE;
       #供料输送机 := TRUE;
       #物料发生器 := TRUE;
   END_IF;
END_REGION

REGION Network 3: 一级停止
   // ，让供料输送机和物料发生器，先停止工作，为了保持在停止或者启动的时候，误按了启动或者停止所有，需要对其进行互锁、
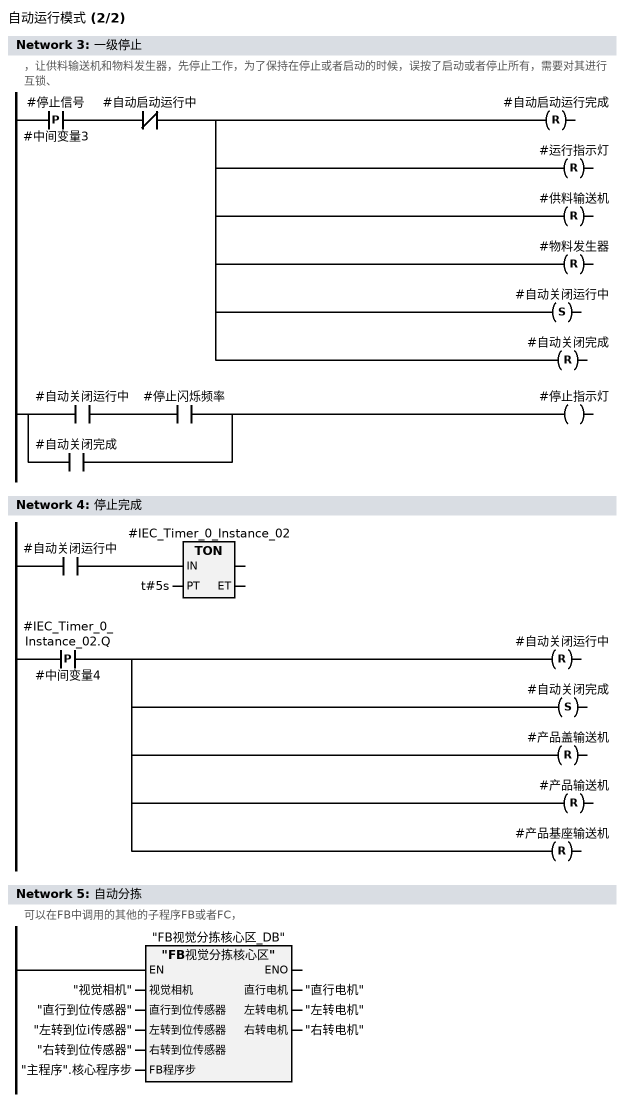
   RUNG wire#powerrail
      P_Contact(operand := #停止信号, bit := #中间变量3)
      I_Contact( #自动启动运行中 )
      wire#w1
      R_Coil( #自动启动运行完成 )
   END_RUNG
   RUNG wire#w1
      R_Coil( #运行指示灯 )
   END_RUNG
   RUNG wire#w1
      R_Coil( #供料输送机 )
   END_RUNG
   RUNG wire#w1
      R_Coil( #物料发生器 )
   END_RUNG
   RUNG wire#w1
      S_Coil( #自动关闭运行中 )
   END_RUNG
   RUNG wire#w1
      R_Coil( #自动关闭完成 )
   END_RUNG
   RUNG wire#powerrail
      Contact( #自动关闭运行中 )
      Contact( #停止闪烁频率 )
      wire#w2
      Coil( #停止指示灯 )
   END_RUNG
   RUNG wire#powerrail
      Contact( #自动关闭完成 )
   END_RUNG wire#w2
   // the same network as SCL:
   #_w1 := #停止信号 AND NOT #中间变量3;   // rising edge of #停止信号
   #中间变量3 := #停止信号;
   IF #_w1 AND NOT #自动启动运行中 THEN
       #自动启动运行完成 := FALSE;
       #运行指示灯 := FALSE;
       #供料输送机 := FALSE;
       #物料发生器 := FALSE;
       #自动关闭运行中 := TRUE;
       #自动关闭完成 := FALSE;
   END_IF;
   #停止指示灯 := (#自动关闭运行中 AND #停止闪烁频率) OR #自动关闭完成;
END_REGION

REGION Network 4: 停止完成
   #IEC_Timer_0_Instance_02(IN := #自动关闭运行中, PT := t#5s);   // TON
   #_w1 := #IEC_Timer_0_Instance_02.Q AND NOT #中间变量4;   // rising edge of #IEC_Timer_0_Instance_02.Q
   #中间变量4 := #IEC_Timer_0_Instance_02.Q;
   IF #_w1 THEN
       #自动关闭运行中 := FALSE;
       #自动关闭完成 := TRUE;
       #产品盖输送机 := FALSE;
       #产品输送机 := FALSE;
       #产品基座输送机 := FALSE;
   END_IF;
END_REGION

REGION Network 5: 自动分拣
   // 可以在FB中调用的其他的子程序FB或者FC，
   RUNG wire#powerrail
      "FB视觉分拣核心区_DB"(视觉相机 := "视觉相机", 直行到位传感器 := "直行到位传感器", 左转到位传感器 := "左转到位i传感器", 右转到位传感器 := "右转到位传感器", FB程序步 := "主程序".核心程序步, 直行电机 => "直行电机", 左转电机 => "左转电机", 右转电机 => "右转电机")
   END_RUNG
   // the same network as SCL:
   "FB视觉分拣核心区_DB"(视觉相机 := "视觉相机",   // "FB视觉分拣核心区"
                  直行到位传感器 := "直行到位传感器",
                  左转到位传感器 := "左转到位i传感器",
                  右转到位传感器 := "右转到位传感器",
                  FB程序步 := "主程序".核心程序步,
                  直行电机 => "直行电机",
                  左转电机 => "左转电机",
                  右转电机 => "右转电机");
END_REGION
END_FUNCTION_BLOCK

// folder: 03_手动运行模式

FUNCTION_BLOCK "手动运行模式"   // FB3, LAD
{ S7_Optimized_Access := 'TRUE' }
VERSION : 0.1
   VAR_INPUT
      启动信号 : Bool;
      停止信号 : Bool;
      复位信号 : Bool;
   END_VAR
   VAR_OUTPUT
      运行指示灯 : Bool;
      复位指示灯 : Bool;
      停止指示灯 : Bool;
      物料发生器 : Bool;
      供料输送机 : Bool;
      产品盖输送机 : Bool;
      产品原料输送机 : Bool;
      产品基座输送机 : Bool;
      阻挡器 : Bool;
   END_VAR
   VAR
      中间变量1 : Bool;
      中间变量2 : Bool;
      中间变量3 : Bool;
      中间变量4 : Bool;
   END_VAR
   VAR_TEMP   // added for the SCL form of the ladder/FBD networks
      _w1 : Bool;
   END_VAR
BEGIN

REGION Network 1: 手动模式下的启动
   // 每次都生成一个物料运输，第二点就是，每一次启动都要将停止信号灯关闭
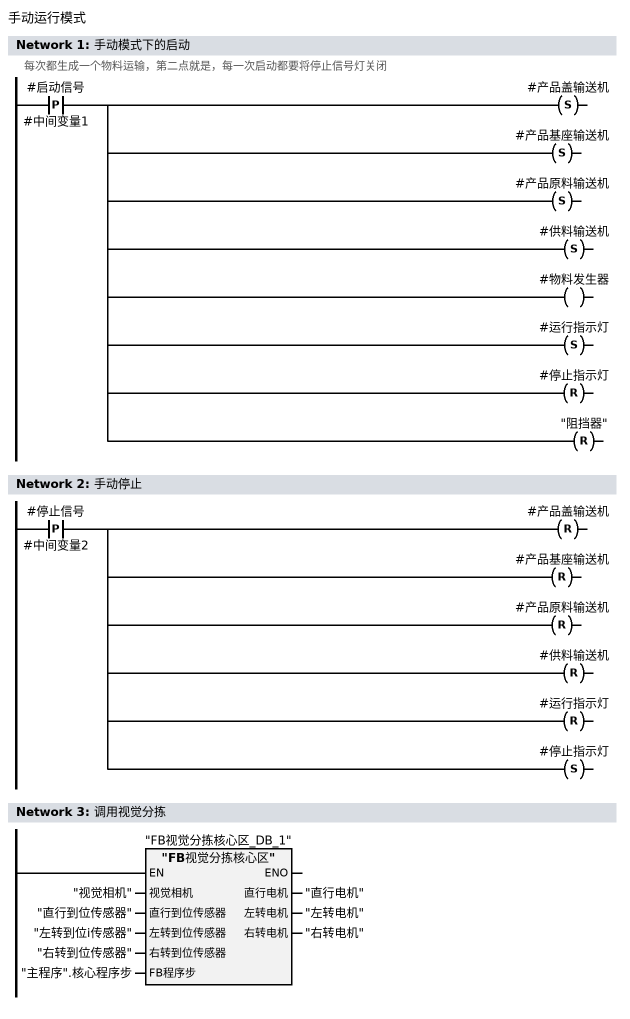
   RUNG wire#powerrail
      P_Contact(operand := #启动信号, bit := #中间变量1)
      wire#w1
      S_Coil( #产品盖输送机 )
   END_RUNG
   RUNG wire#w1
      S_Coil( #产品基座输送机 )
   END_RUNG
   RUNG wire#w1
      S_Coil( #产品原料输送机 )
   END_RUNG
   RUNG wire#w1
      S_Coil( #供料输送机 )
   END_RUNG
   RUNG wire#w1
      Coil( #物料发生器 )
   END_RUNG
   RUNG wire#w1
      S_Coil( #运行指示灯 )
   END_RUNG
   RUNG wire#w1
      R_Coil( #停止指示灯 )
   END_RUNG
   RUNG wire#w1
      R_Coil( "阻挡器" )
   END_RUNG
   // the same network as SCL:
   #_w1 := #启动信号 AND NOT #中间变量1;   // rising edge of #启动信号
   #中间变量1 := #启动信号;
   IF #_w1 THEN
       #产品盖输送机 := TRUE;
       #产品基座输送机 := TRUE;
       #产品原料输送机 := TRUE;
       #供料输送机 := TRUE;
   END_IF;
   #物料发生器 := #_w1;
   IF #_w1 THEN
       #运行指示灯 := TRUE;
       #停止指示灯 := FALSE;
       "阻挡器" := FALSE;
   END_IF;
END_REGION

REGION Network 2: 手动停止
   RUNG wire#powerrail
      P_Contact(operand := #停止信号, bit := #中间变量2)
      wire#w1
      R_Coil( #产品盖输送机 )
   END_RUNG
   RUNG wire#w1
      R_Coil( #产品基座输送机 )
   END_RUNG
   RUNG wire#w1
      R_Coil( #产品原料输送机 )
   END_RUNG
   RUNG wire#w1
      R_Coil( #供料输送机 )
   END_RUNG
   RUNG wire#w1
      R_Coil( #运行指示灯 )
   END_RUNG
   RUNG wire#w1
      S_Coil( #停止指示灯 )
   END_RUNG
   // the same network as SCL:
   #_w1 := #停止信号 AND NOT #中间变量2;   // rising edge of #停止信号
   #中间变量2 := #停止信号;
   IF #_w1 THEN
       #产品盖输送机 := FALSE;
       #产品基座输送机 := FALSE;
       #产品原料输送机 := FALSE;
       #供料输送机 := FALSE;
       #运行指示灯 := FALSE;
       #停止指示灯 := TRUE;
   END_IF;
END_REGION

REGION Network 3: 调用视觉分拣
   RUNG wire#powerrail
      "FB视觉分拣核心区_DB_1"(视觉相机 := "视觉相机", 直行到位传感器 := "直行到位传感器", 左转到位传感器 := "左转到位i传感器", 右转到位传感器 := "右转到位传感器", FB程序步 := "主程序".核心程序步, 直行电机 => "直行电机", 左转电机 => "左转电机", 右转电机 => "右转电机")
   END_RUNG
   // the same network as SCL:
   "FB视觉分拣核心区_DB_1"(视觉相机 := "视觉相机",   // "FB视觉分拣核心区"
                    直行到位传感器 := "直行到位传感器",
                    左转到位传感器 := "左转到位i传感器",
                    右转到位传感器 := "右转到位传感器",
                    FB程序步 := "主程序".核心程序步,
                    直行电机 => "直行电机",
                    左转电机 => "左转电机",
                    右转电机 => "右转电机");
END_REGION
END_FUNCTION_BLOCK

// folder: 04_系统急停

FUNCTION_BLOCK "系统急停"   // FB4, LAD
{ S7_Optimized_Access := 'TRUE' }
VERSION : 0.1
   VAR_INPUT
      急停闪烁按钮 : Bool;
   END_VAR
   VAR_OUTPUT
      供料输送机 : Bool;
      物料发生器 : Bool;
      直行电机 : Bool;
      左转电机 : Bool;
      右转电机 : Bool;
      产品原料输送机 : Bool;
      产品盖输送机 : Bool;
      产品基座输送机 : Bool;
      运行指示灯 : Bool;
      停止指示灯 : Bool;
      阻挡器 : Bool;
      复位指示灯 : Bool;
   END_VAR
BEGIN

REGION Network 1
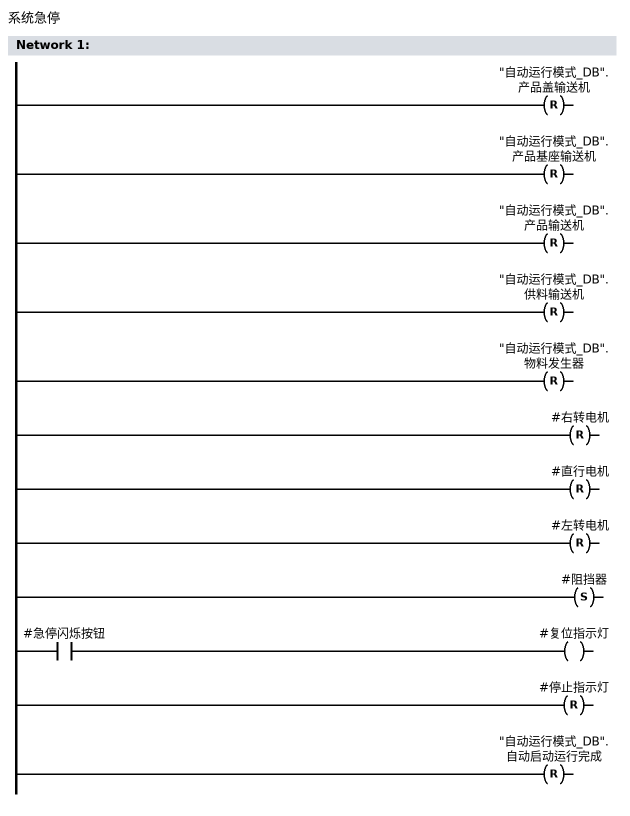
   RUNG wire#powerrail
      R_Coil( "自动运行模式_DB".产品盖输送机 )
   END_RUNG
   RUNG wire#powerrail
      R_Coil( "自动运行模式_DB".产品基座输送机 )
   END_RUNG
   RUNG wire#powerrail
      R_Coil( "自动运行模式_DB".产品输送机 )
   END_RUNG
   RUNG wire#powerrail
      R_Coil( "自动运行模式_DB".供料输送机 )
   END_RUNG
   RUNG wire#powerrail
      R_Coil( "自动运行模式_DB".物料发生器 )
   END_RUNG
   RUNG wire#powerrail
      R_Coil( #右转电机 )
   END_RUNG
   RUNG wire#powerrail
      R_Coil( #直行电机 )
   END_RUNG
   RUNG wire#powerrail
      R_Coil( #左转电机 )
   END_RUNG
   RUNG wire#powerrail
      S_Coil( #阻挡器 )
   END_RUNG
   RUNG wire#powerrail
      Contact( #急停闪烁按钮 )
      Coil( #复位指示灯 )
   END_RUNG
   RUNG wire#powerrail
      R_Coil( #停止指示灯 )
   END_RUNG
   RUNG wire#powerrail
      R_Coil( "自动运行模式_DB".自动启动运行完成 )
   END_RUNG
   // the same network as SCL:
   "自动运行模式_DB".产品盖输送机 := FALSE;
   "自动运行模式_DB".产品基座输送机 := FALSE;
   "自动运行模式_DB".产品输送机 := FALSE;
   "自动运行模式_DB".供料输送机 := FALSE;
   "自动运行模式_DB".物料发生器 := FALSE;
   #右转电机 := FALSE;
   #直行电机 := FALSE;
   #左转电机 := FALSE;
   #阻挡器 := TRUE;
   #复位指示灯 := #急停闪烁按钮;
   #停止指示灯 := FALSE;
   "自动运行模式_DB".自动启动运行完成 := FALSE;
END_REGION
END_FUNCTION_BLOCK

// folder: 05_系统复位

FUNCTION_BLOCK "系统复位"   // FB5, LAD
{ S7_Optimized_Access := 'TRUE' }
VERSION : 0.1
   VAR
      IEC_Timer_0_Instance : TON_TIME;
      中间变量1 : Bool;
      中间变量2 : Bool;
      中间变量3 : Bool;
      中间变量4 : Bool;
   END_VAR
   VAR_TEMP   // added for the SCL form of the ladder/FBD networks
      _w1 : Bool;
   END_VAR
BEGIN

REGION Network 1: 复位
   // 为了避免调用FB块时，DB的输出对于IO表的控制，再复位中我们选择IO表达输出直接当输出
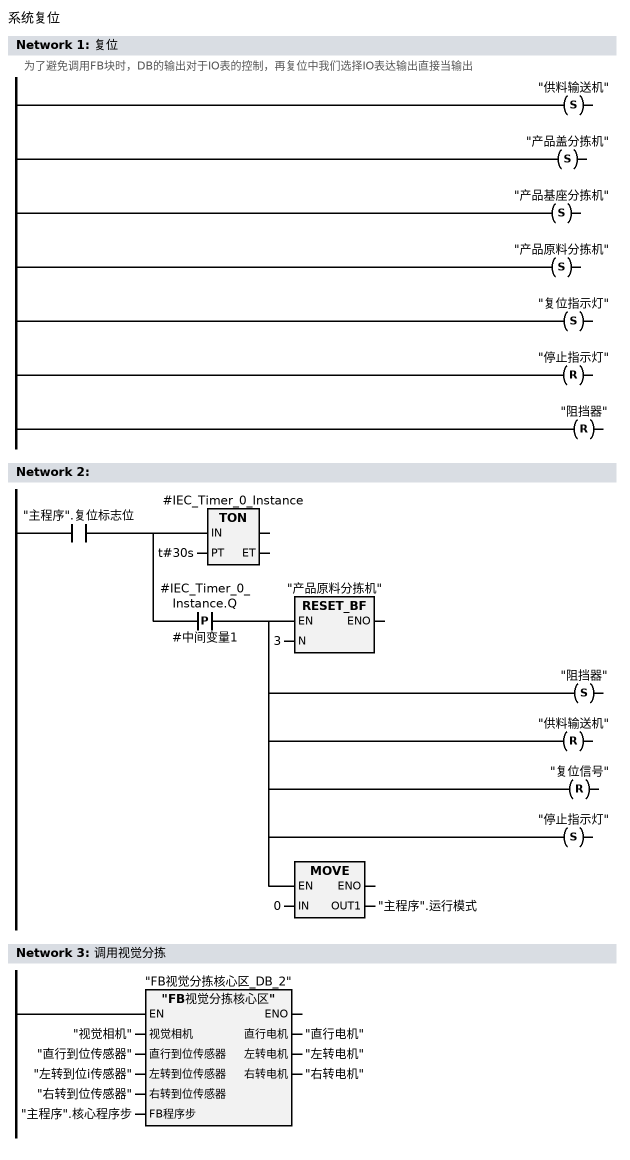
   RUNG wire#powerrail
      S_Coil( "供料输送机" )
   END_RUNG
   RUNG wire#powerrail
      S_Coil( "产品盖分拣机" )
   END_RUNG
   RUNG wire#powerrail
      S_Coil( "产品基座分拣机" )
   END_RUNG
   RUNG wire#powerrail
      S_Coil( "产品原料分拣机" )
   END_RUNG
   RUNG wire#powerrail
      S_Coil( "复位指示灯" )
   END_RUNG
   RUNG wire#powerrail
      R_Coil( "停止指示灯" )
   END_RUNG
   RUNG wire#powerrail
      R_Coil( "阻挡器" )
   END_RUNG
   // the same network as SCL:
   "供料输送机" := TRUE;
   "产品盖分拣机" := TRUE;
   "产品基座分拣机" := TRUE;
   "产品原料分拣机" := TRUE;
   "复位指示灯" := TRUE;
   "停止指示灯" := FALSE;
   "阻挡器" := FALSE;
END_REGION

REGION Network 2
   // no SCL statement known for RBitfield: written as a call
   #IEC_Timer_0_Instance(IN := "主程序".复位标志位, PT := t#30s);   // TON
   #_w1 := "主程序".复位标志位 AND #IEC_Timer_0_Instance.Q AND NOT #中间变量1;   // rising edge of #IEC_Timer_0_Instance.Q
   #中间变量1 := #IEC_Timer_0_Instance.Q;
   IF #_w1 THEN
       RESET_BF(operand := "产品原料分拣机", n := 3);
       "阻挡器" := TRUE;
       "供料输送机" := FALSE;
       "复位信号" := FALSE;
       "停止指示灯" := TRUE;
       "主程序".运行模式 := 0;
   END_IF;
END_REGION

REGION Network 3: 调用视觉分拣
   RUNG wire#powerrail
      "FB视觉分拣核心区_DB_2"(视觉相机 := "视觉相机", 直行到位传感器 := "直行到位传感器", 左转到位传感器 := "左转到位i传感器", 右转到位传感器 := "右转到位传感器", FB程序步 := "主程序".核心程序步, 直行电机 => "直行电机", 左转电机 => "左转电机", 右转电机 => "右转电机")
   END_RUNG
   // the same network as SCL:
   "FB视觉分拣核心区_DB_2"(视觉相机 := "视觉相机",   // "FB视觉分拣核心区"
                    直行到位传感器 := "直行到位传感器",
                    左转到位传感器 := "左转到位i传感器",
                    右转到位传感器 := "右转到位传感器",
                    FB程序步 := "主程序".核心程序步,
                    直行电机 => "直行电机",
                    左转电机 => "左转电机",
                    右转电机 => "右转电机");
END_REGION
END_FUNCTION_BLOCK

(* ===== HMI "HMI_RT_1" =====
system functions are stored by id; their names below are inferred from use
connection "HMI_连接_1": ETHERNET, SMART_S7_1200_OMS

HMI tags "默认变量表"
   "Tag_ScreenNumber" : UInt, internal
   "主程序_手/自动切换" : Bool = PLC 主程序.手/自动切换, 1 s
   "主程序_急停信号" : Bool = PLC 主程序.急停信号, 1 s
   "主程序_启动信号" : Bool = PLC 主程序.启动信号, 1 s
   "主程序_停止信号" : Bool = PLC 主程序.停止信号, 1 s
   "主程序_复位信号" : Bool = PLC 主程序.复位信号, 1 s

Template "模板_1" 800x480
   Button "退出" at 714,429 size 71x50; TextOff '退出'; PictureOff "ExitRuntime_KTP700_Basic_PN_TR"; PictureOn "ExitRuntime_KTP700_Basic_PN_TR"
      on Release: StopRuntime(0)
   Button "Template_Button" at 614,429 size 71x50; TextOff 'Text'
   Button "Template_Button_1" at 514,429 size 71x50; TextOff 'Text'
   Button "Template_Button_2" at 414,429 size 71x50; TextOff 'Text'
   Button "Template_Button_3" at 314,429 size 71x50; TextOff 'Text'
   Button "Template_Button_4" at 214,429 size 71x50; TextOff 'Text'
   Button "Template_Button_5" at 114,429 size 71x50; TextOff 'Text'
   Button "起始画面" at 14,429 size 71x50; TextOff '起始画面'; PictureOff "NavigateHome_KTP700_Basic_PN_TR"; PictureOn "NavigateHome_KTP700_Basic_PN_TR"
      on Release: ActivateScreen("根画面", 0)
   SymbolicIOField "Symbolic_IO_Field_Screen" at 93,9 size 600x33; TextOff '0'; TextOn '1'; TextList "TextList_ScreenNames"
      ProcessValue <- "Tag_ScreenNumber"
      on Change: ActivateScreenByNumber("Tag_ScreenNumber", 0)
   DateTimeField "HmiScreenItemData" at 695,25 size 105x25
   DateTimeField "HmiScreenItemData_1" at 695,0 size 105x25
   GraphicView "Logo" at 0,0 size 91x51; Picture "HMI_1 的 Logo"

screen "根画面" 800x480, template "模板_1"
   on GenerateScreen: SetTag("Tag_ScreenNumber", 1)
   TextField "文本域_1" at 293,41 size 203x37; Text '视觉分拣练习'
   Switch "开关_1" at 123,139 size 96x36; CaptionText 'Switch'; TextOff '手动'; TextOn '自动'
      ProcessValue <- "主程序_手/自动切换"
   Button "按钮_1" at 123,232 size 96x37; TextOff '急停'
      on Click: InvertBit("主程序_急停信号")
   Button "按钮_2" at 608,136 size 96x37; TextOff '启动'
      on Press: SetBit("主程序_启动信号")
      on Release: ResetBit("主程序_启动信号")
   Button "按钮_3" at 608,225 size 96x37; TextOff '停止'
      on Release: ResetBit("主程序_停止信号")
      on Press: SetBit("主程序_停止信号")
   Button "按钮_4" at 608,318 size 96x37; TextOff '复位'
      on Press: SetBit("主程序_复位信号")
      on Release: ResetBit("主程序_复位信号")
*)